// TIA Portal V20 export
// export: Created 2026-07-10T11:12:27.9543824Z, ExportSetting WithDefaults, DisplayName Totally Integrated Automation Portal, DisplayVersion V20, DisplayName TIA Portal Openness, DisplayVersion V20, DisplayName TIA Portal Version Control Interface, DisplayVersion V20, DisplayName STEP 7 Professional, DisplayVersion V20, DisplayName STEP 7 Safety, DisplayVersion V20, DisplayName WinCC Basic/Comfort/Advanced, DisplayVersion V20, DisplayName WinCC Unified, DisplayVersion V20
DATA_BLOCK "Weighting_DB"   // DB12
VERSION : 0.1
// stored: AutoNumber true, DBAccessibleFromOPCUA true, InstanceOfName Weighting, InstanceOfType FB
"Weighting"
   // VAR
   //    buffer1 { S7_SetPoint := 'True'} : Array[0..1] of Word;
   //    buffer2 : Array[0..1] of Word;
   //    Enable { S7_SetPoint := 'True'} : Bool;
   //    ManualValueProvided1 : Bool;
   //    ManualValueProvided2 : Bool;
   //    ManualValue1 : Real;
   //    ManualValue2 : Real;
   //    WeightHandlers : Array[0..1] of "WeightHandler";
   //    TankWeigher1 { S7_SetPoint := 'True'} : "TankWeigher";
   //    RetainData : "WeightRetainData";
   //    TimeNow { S7_SetPoint := 'True'} : DTL;
   // END_VAR
BEGIN
   buffer1[0..1] := 16#0000;
END_DATA_BLOCK
